{attribute 'qualified_only'}
{attribute 'to_string'}
TYPE ST110_PnpHorPos_e :
(
	GS,
	AS,
	_max
);
END_TYPE

(* stored: Version 1.1.0.1, ProductVersion 3.1.4024.6
   DUT ST110_PnpHorPos_e: Id {84e1a7e3-96fd-41b8-9875-96adbe80b49b} *)
